FUNCTION F_Convert10V2Temp : INT
VAR_INPUT
	i_Value			:	INT;
END_VAR
VAR_OUTPUT
END_VAR
VAR
	r_converted2V 	: 	REAL;
	i_finalValue	:	INT;
END_VAR

// For Convertion of 0-10V Signal from 0-50°C

r_converted2V := i_Value * 0.00030518509476;
i_finalValue := REAL_TO_INT((r_converted2V / 2) * 100);

F_Convert10V2Temp := i_finalValue;

END_FUNCTION

(* stored: Version 1.1.0.1, ProductVersion 3.1.4024.4
   POU F_Convert10V2Temp: Id {cf8c24de-51eb-467f-b321-46e2aa96626e}, SpecialFunc None *)
